// TIA Portal V16 export
// export: Created 2022-09-01T14:29:20.4817445Z, ExportSetting WithDefaults, DisplayName Totally Integrated Automation Portal, DisplayVersion V16, DisplayName TIA Portal Version Control Interface, DisplayVersion V16, DisplayName TIA Portal Openness, DisplayVersion V16, DisplayName STEP 7 Professional, DisplayVersion V16, DisplayName STEP 7 Safety, DisplayVersion V16, DisplayName WinCC Advanced, DisplayVersion V16
FUNCTION "Saídas" : Void   // FC2, LAD
{ S7_Optimized_Access := 'TRUE' }
VERSION : 0.1
// stored: AutoNumber true, IsIECCheckEnabled false, SetENOAutomatically false, UDAEnableTagReadback false
   VAR_TEMP   // added for the SCL form of the ladder/FBD networks
      _w1 : Bool;
   END_VAR
BEGIN

REGION Network 1: bomba de alimentação ao processo BS001A
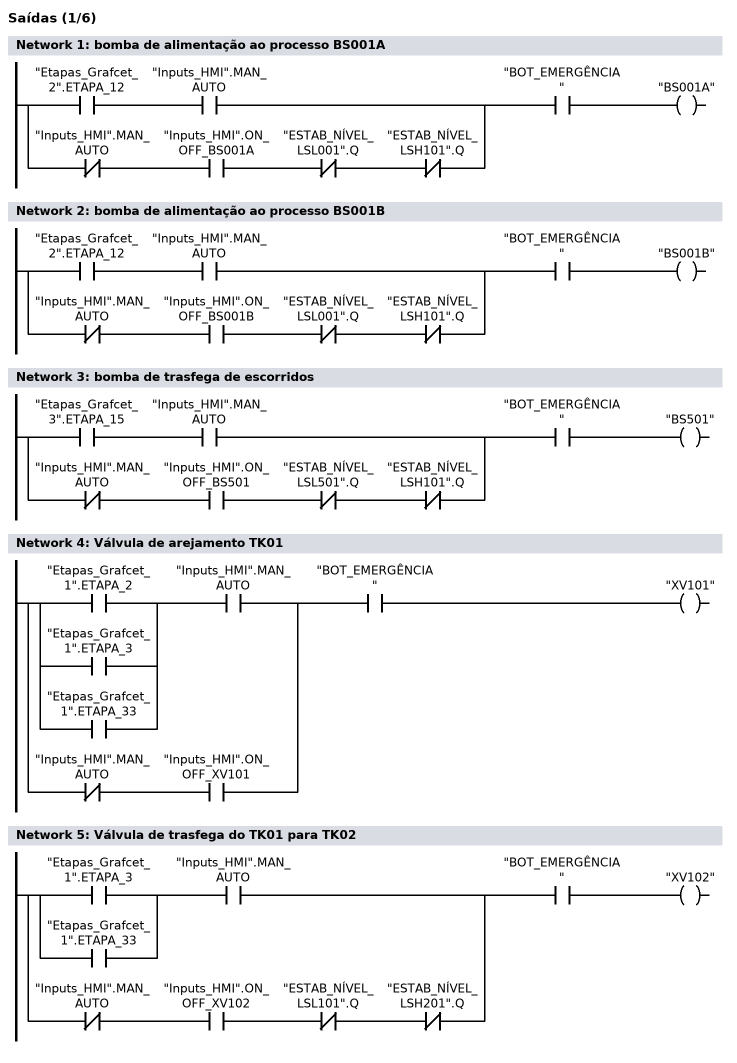
   RUNG wire#powerrail
      Contact( "Etapas_Grafcet_2".ETAPA_12 )
      Contact( "Inputs_HMI".MAN_AUTO )
      wire#w1
      Contact( "BOT_EMERGÊNCIA" )
      Coil( "BS001A" )
   END_RUNG
   RUNG wire#powerrail
      I_Contact( "Inputs_HMI".MAN_AUTO )
      Contact( "Inputs_HMI".ON_OFF_BS001A )
      I_Contact( "ESTAB_NÍVEL_LSL001".Q )
      I_Contact( "ESTAB_NÍVEL_LSH101".Q )
   END_RUNG wire#w1
   // the same network as SCL:
   "BS001A" := (("Etapas_Grafcet_2".ETAPA_12 AND "Inputs_HMI".MAN_AUTO) OR (NOT "Inputs_HMI".MAN_AUTO AND "Inputs_HMI".ON_OFF_BS001A AND NOT "ESTAB_NÍVEL_LSL001".Q AND NOT "ESTAB_NÍVEL_LSH101".Q)) AND "BOT_EMERGÊNCIA";
END_REGION

REGION Network 2: bomba de alimentação ao processo BS001B
   RUNG wire#powerrail
      Contact( "Etapas_Grafcet_2".ETAPA_12 )
      Contact( "Inputs_HMI".MAN_AUTO )
      wire#w1
      Contact( "BOT_EMERGÊNCIA" )
      Coil( "BS001B" )
   END_RUNG
   RUNG wire#powerrail
      I_Contact( "Inputs_HMI".MAN_AUTO )
      Contact( "Inputs_HMI".ON_OFF_BS001B )
      I_Contact( "ESTAB_NÍVEL_LSL001".Q )
      I_Contact( "ESTAB_NÍVEL_LSH101".Q )
   END_RUNG wire#w1
   // the same network as SCL:
   "BS001B" := (("Etapas_Grafcet_2".ETAPA_12 AND "Inputs_HMI".MAN_AUTO) OR (NOT "Inputs_HMI".MAN_AUTO AND "Inputs_HMI".ON_OFF_BS001B AND NOT "ESTAB_NÍVEL_LSL001".Q AND NOT "ESTAB_NÍVEL_LSH101".Q)) AND "BOT_EMERGÊNCIA";
END_REGION

REGION Network 3: bomba de trasfega de escorridos
   RUNG wire#powerrail
      Contact( "Etapas_Grafcet_3".ETAPA_15 )
      Contact( "Inputs_HMI".MAN_AUTO )
      wire#w1
      Contact( "BOT_EMERGÊNCIA" )
      Coil( "BS501" )
   END_RUNG
   RUNG wire#powerrail
      I_Contact( "Inputs_HMI".MAN_AUTO )
      Contact( "Inputs_HMI".ON_OFF_BS501 )
      I_Contact( "ESTAB_NÍVEL_LSL501".Q )
      I_Contact( "ESTAB_NÍVEL_LSH101".Q )
   END_RUNG wire#w1
   // the same network as SCL:
   "BS501" := (("Etapas_Grafcet_3".ETAPA_15 AND "Inputs_HMI".MAN_AUTO) OR (NOT "Inputs_HMI".MAN_AUTO AND "Inputs_HMI".ON_OFF_BS501 AND NOT "ESTAB_NÍVEL_LSL501".Q AND NOT "ESTAB_NÍVEL_LSH101".Q)) AND "BOT_EMERGÊNCIA";
END_REGION

REGION Network 4: Válvula de arejamento TK01
   RUNG wire#powerrail
      Contact( "Etapas_Grafcet_1".ETAPA_2 )
      wire#w1
      Contact( "Inputs_HMI".MAN_AUTO )
      wire#w2
      Contact( "BOT_EMERGÊNCIA" )
      Coil( "XV101" )
   END_RUNG
   RUNG wire#powerrail
      Contact( "Etapas_Grafcet_1".ETAPA_3 )
   END_RUNG wire#w1
   RUNG wire#powerrail
      Contact( "Etapas_Grafcet_1".ETAPA_33 )
   END_RUNG wire#w1
   RUNG wire#powerrail
      I_Contact( "Inputs_HMI".MAN_AUTO )
      Contact( "Inputs_HMI".ON_OFF_XV101 )
   END_RUNG wire#w2
   // the same network as SCL:
   "XV101" := ((("Etapas_Grafcet_1".ETAPA_2 OR "Etapas_Grafcet_1".ETAPA_3 OR "Etapas_Grafcet_1".ETAPA_33) AND "Inputs_HMI".MAN_AUTO) OR (NOT "Inputs_HMI".MAN_AUTO AND "Inputs_HMI".ON_OFF_XV101)) AND "BOT_EMERGÊNCIA";
END_REGION

REGION Network 5: Válvula de trasfega do TK01 para TK02
   RUNG wire#powerrail
      Contact( "Etapas_Grafcet_1".ETAPA_3 )
      wire#w1
      Contact( "Inputs_HMI".MAN_AUTO )
      wire#w2
      Contact( "BOT_EMERGÊNCIA" )
      Coil( "XV102" )
   END_RUNG
   RUNG wire#powerrail
      Contact( "Etapas_Grafcet_1".ETAPA_33 )
   END_RUNG wire#w1
   RUNG wire#powerrail
      I_Contact( "Inputs_HMI".MAN_AUTO )
      Contact( "Inputs_HMI".ON_OFF_XV102 )
      I_Contact( "ESTAB_NÍVEL_LSL101".Q )
      I_Contact( "ESTAB_NÍVEL_LSH201".Q )
   END_RUNG wire#w2
   // the same network as SCL:
   "XV102" := ((("Etapas_Grafcet_1".ETAPA_3 OR "Etapas_Grafcet_1".ETAPA_33) AND "Inputs_HMI".MAN_AUTO) OR (NOT "Inputs_HMI".MAN_AUTO AND "Inputs_HMI".ON_OFF_XV102 AND NOT "ESTAB_NÍVEL_LSL101".Q AND NOT "ESTAB_NÍVEL_LSH201".Q)) AND "BOT_EMERGÊNCIA";
END_REGION

REGION Network 6: Agitador MX201
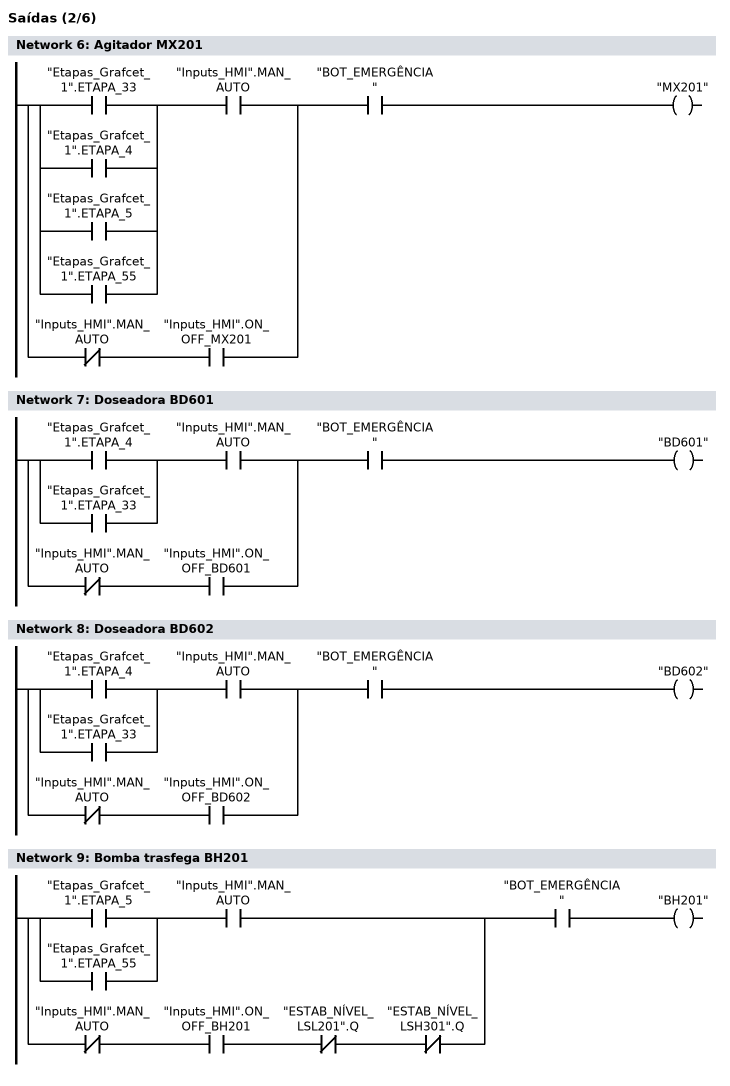
   RUNG wire#powerrail
      Contact( "Etapas_Grafcet_1".ETAPA_33 )
      wire#w1
      Contact( "Inputs_HMI".MAN_AUTO )
      wire#w2
      Contact( "BOT_EMERGÊNCIA" )
      Coil( "MX201" )
   END_RUNG
   RUNG wire#powerrail
      Contact( "Etapas_Grafcet_1".ETAPA_4 )
   END_RUNG wire#w1
   RUNG wire#powerrail
      Contact( "Etapas_Grafcet_1".ETAPA_5 )
   END_RUNG wire#w1
   RUNG wire#powerrail
      Contact( "Etapas_Grafcet_1".ETAPA_55 )
   END_RUNG wire#w1
   RUNG wire#powerrail
      I_Contact( "Inputs_HMI".MAN_AUTO )
      Contact( "Inputs_HMI".ON_OFF_MX201 )
   END_RUNG wire#w2
   // the same network as SCL:
   "MX201" := ((("Etapas_Grafcet_1".ETAPA_33 OR "Etapas_Grafcet_1".ETAPA_4 OR "Etapas_Grafcet_1".ETAPA_5 OR "Etapas_Grafcet_1".ETAPA_55) AND "Inputs_HMI".MAN_AUTO) OR (NOT "Inputs_HMI".MAN_AUTO AND "Inputs_HMI".ON_OFF_MX201)) AND "BOT_EMERGÊNCIA";
END_REGION

REGION Network 7: Doseadora BD601
   RUNG wire#powerrail
      Contact( "Etapas_Grafcet_1".ETAPA_4 )
      wire#w1
      Contact( "Inputs_HMI".MAN_AUTO )
      wire#w2
      Contact( "BOT_EMERGÊNCIA" )
      Coil( "BD601" )
   END_RUNG
   RUNG wire#powerrail
      Contact( "Etapas_Grafcet_1".ETAPA_33 )
   END_RUNG wire#w1
   RUNG wire#powerrail
      I_Contact( "Inputs_HMI".MAN_AUTO )
      Contact( "Inputs_HMI".ON_OFF_BD601 )
   END_RUNG wire#w2
   // the same network as SCL:
   "BD601" := ((("Etapas_Grafcet_1".ETAPA_4 OR "Etapas_Grafcet_1".ETAPA_33) AND "Inputs_HMI".MAN_AUTO) OR (NOT "Inputs_HMI".MAN_AUTO AND "Inputs_HMI".ON_OFF_BD601)) AND "BOT_EMERGÊNCIA";
END_REGION

REGION Network 8: Doseadora BD602
   RUNG wire#powerrail
      Contact( "Etapas_Grafcet_1".ETAPA_4 )
      wire#w1
      Contact( "Inputs_HMI".MAN_AUTO )
      wire#w2
      Contact( "BOT_EMERGÊNCIA" )
      Coil( "BD602" )
   END_RUNG
   RUNG wire#powerrail
      Contact( "Etapas_Grafcet_1".ETAPA_33 )
   END_RUNG wire#w1
   RUNG wire#powerrail
      I_Contact( "Inputs_HMI".MAN_AUTO )
      Contact( "Inputs_HMI".ON_OFF_BD602 )
   END_RUNG wire#w2
   // the same network as SCL:
   "BD602" := ((("Etapas_Grafcet_1".ETAPA_4 OR "Etapas_Grafcet_1".ETAPA_33) AND "Inputs_HMI".MAN_AUTO) OR (NOT "Inputs_HMI".MAN_AUTO AND "Inputs_HMI".ON_OFF_BD602)) AND "BOT_EMERGÊNCIA";
END_REGION

REGION Network 9: Bomba trasfega BH201
   RUNG wire#powerrail
      Contact( "Etapas_Grafcet_1".ETAPA_5 )
      wire#w1
      Contact( "Inputs_HMI".MAN_AUTO )
      wire#w2
      Contact( "BOT_EMERGÊNCIA" )
      Coil( "BH201" )
   END_RUNG
   RUNG wire#powerrail
      Contact( "Etapas_Grafcet_1".ETAPA_55 )
   END_RUNG wire#w1
   RUNG wire#powerrail
      I_Contact( "Inputs_HMI".MAN_AUTO )
      Contact( "Inputs_HMI".ON_OFF_BH201 )
      I_Contact( "ESTAB_NÍVEL_LSL201".Q )
      I_Contact( "ESTAB_NÍVEL_LSH301".Q )
   END_RUNG wire#w2
   // the same network as SCL:
   "BH201" := ((("Etapas_Grafcet_1".ETAPA_5 OR "Etapas_Grafcet_1".ETAPA_55) AND "Inputs_HMI".MAN_AUTO) OR (NOT "Inputs_HMI".MAN_AUTO AND "Inputs_HMI".ON_OFF_BH201 AND NOT "ESTAB_NÍVEL_LSL201".Q AND NOT "ESTAB_NÍVEL_LSH301".Q)) AND "BOT_EMERGÊNCIA";
END_REGION

REGION Network 10: Agitador MX301
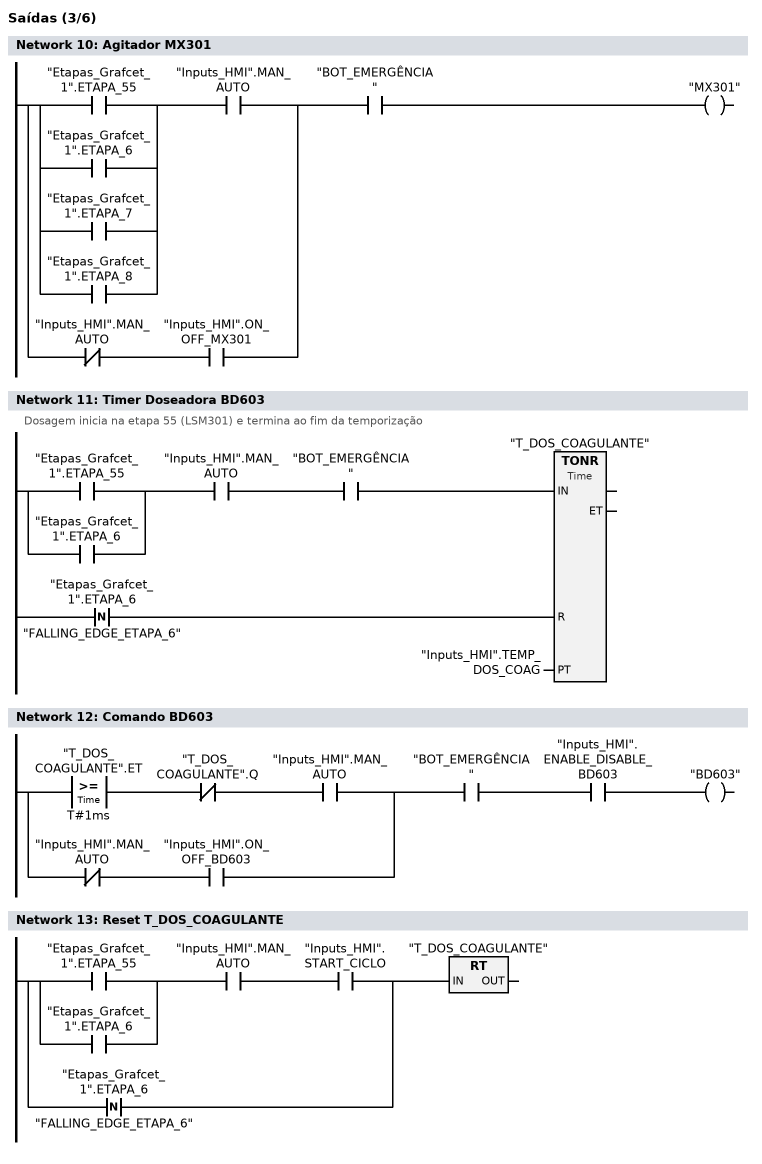
   RUNG wire#powerrail
      Contact( "Etapas_Grafcet_1".ETAPA_55 )
      wire#w1
      Contact( "Inputs_HMI".MAN_AUTO )
      wire#w2
      Contact( "BOT_EMERGÊNCIA" )
      Coil( "MX301" )
   END_RUNG
   RUNG wire#powerrail
      Contact( "Etapas_Grafcet_1".ETAPA_6 )
   END_RUNG wire#w1
   RUNG wire#powerrail
      Contact( "Etapas_Grafcet_1".ETAPA_7 )
   END_RUNG wire#w1
   RUNG wire#powerrail
      Contact( "Etapas_Grafcet_1".ETAPA_8 )
   END_RUNG wire#w1
   RUNG wire#powerrail
      I_Contact( "Inputs_HMI".MAN_AUTO )
      Contact( "Inputs_HMI".ON_OFF_MX301 )
   END_RUNG wire#w2
   // the same network as SCL:
   "MX301" := ((("Etapas_Grafcet_1".ETAPA_55 OR "Etapas_Grafcet_1".ETAPA_6 OR "Etapas_Grafcet_1".ETAPA_7 OR "Etapas_Grafcet_1".ETAPA_8) AND "Inputs_HMI".MAN_AUTO) OR (NOT "Inputs_HMI".MAN_AUTO AND "Inputs_HMI".ON_OFF_MX301)) AND "BOT_EMERGÊNCIA";
END_REGION

REGION Network 11: Timer Doseadora BD603
   // Dosagem inicia na etapa 55 (LSM301) e termina ao fim da temporização
   RUNG wire#powerrail
      Contact( "Etapas_Grafcet_1".ETAPA_55 )
      wire#w1
      Contact( "Inputs_HMI".MAN_AUTO )
      Contact( "BOT_EMERGÊNCIA" )
      { S7_Templates := "time_type := Time" } "T_DOS_COAGULANTE".TONR(r := wire#w2, pt := "Inputs_HMI".TEMP_DOS_COAG, et =>)
   END_RUNG
   RUNG wire#powerrail
      Contact( "Etapas_Grafcet_1".ETAPA_6 )
   END_RUNG wire#w1
   RUNG wire#powerrail
      N_Contact(operand := "Etapas_Grafcet_1".ETAPA_6, bit := "FALLING_EDGE_ETAPA_6")
   END_RUNG wire#w2
   // the same network as SCL:
   #_w1 := NOT "Etapas_Grafcet_1".ETAPA_6 AND "FALLING_EDGE_ETAPA_6";   // falling edge of "Etapas_Grafcet_1".ETAPA_6
   "FALLING_EDGE_ETAPA_6" := "Etapas_Grafcet_1".ETAPA_6;
   "T_DOS_COAGULANTE".TONR(IN := ("Etapas_Grafcet_1".ETAPA_55 OR "Etapas_Grafcet_1".ETAPA_6) AND "Inputs_HMI".MAN_AUTO AND "BOT_EMERGÊNCIA",
                           R := #_w1,
                           PT := "Inputs_HMI".TEMP_DOS_COAG);
END_REGION

REGION Network 12: Comando BD603
   RUNG wire#powerrail
      { S7_Templates := "SrcType := Time" } GE_Contact(in1 := "T_DOS_COAGULANTE".ET, in2 := T#1ms)
      I_Contact( "T_DOS_COAGULANTE".Q )
      Contact( "Inputs_HMI".MAN_AUTO )
      wire#w1
      Contact( "BOT_EMERGÊNCIA" )
      Contact( "Inputs_HMI".ENABLE_DISABLE_BD603 )
      Coil( "BD603" )
   END_RUNG
   RUNG wire#powerrail
      I_Contact( "Inputs_HMI".MAN_AUTO )
      Contact( "Inputs_HMI".ON_OFF_BD603 )
   END_RUNG wire#w1
   // the same network as SCL:
   "BD603" := ((("T_DOS_COAGULANTE".ET >= T#1ms) AND NOT "T_DOS_COAGULANTE".Q AND "Inputs_HMI".MAN_AUTO) OR (NOT "Inputs_HMI".MAN_AUTO AND "Inputs_HMI".ON_OFF_BD603)) AND "BOT_EMERGÊNCIA" AND "Inputs_HMI".ENABLE_DISABLE_BD603;
END_REGION

REGION Network 13: Reset T_DOS_COAGULANTE
   RUNG wire#powerrail
      Contact( "Etapas_Grafcet_1".ETAPA_55 )
      wire#w1
      Contact( "Inputs_HMI".MAN_AUTO )
      Contact( "Inputs_HMI".START_CICLO )
      wire#w2
      RT_Coil( "T_DOS_COAGULANTE" )
   END_RUNG
   RUNG wire#powerrail
      Contact( "Etapas_Grafcet_1".ETAPA_6 )
   END_RUNG wire#w1
   RUNG wire#powerrail
      N_Contact(operand := "Etapas_Grafcet_1".ETAPA_6, bit := "FALLING_EDGE_ETAPA_6")
   END_RUNG wire#w2
   // the same network as SCL:
   #_w1 := NOT "Etapas_Grafcet_1".ETAPA_6 AND "FALLING_EDGE_ETAPA_6";   // falling edge of "Etapas_Grafcet_1".ETAPA_6
   "FALLING_EDGE_ETAPA_6" := "Etapas_Grafcet_1".ETAPA_6;
   IF (("Etapas_Grafcet_1".ETAPA_55 OR "Etapas_Grafcet_1".ETAPA_6) AND "Inputs_HMI".MAN_AUTO AND "Inputs_HMI".START_CICLO) OR #_w1 THEN
       RESET_TIMER("T_DOS_COAGULANTE");
   END_IF;
END_REGION

REGION Network 14: Doseadora BD604
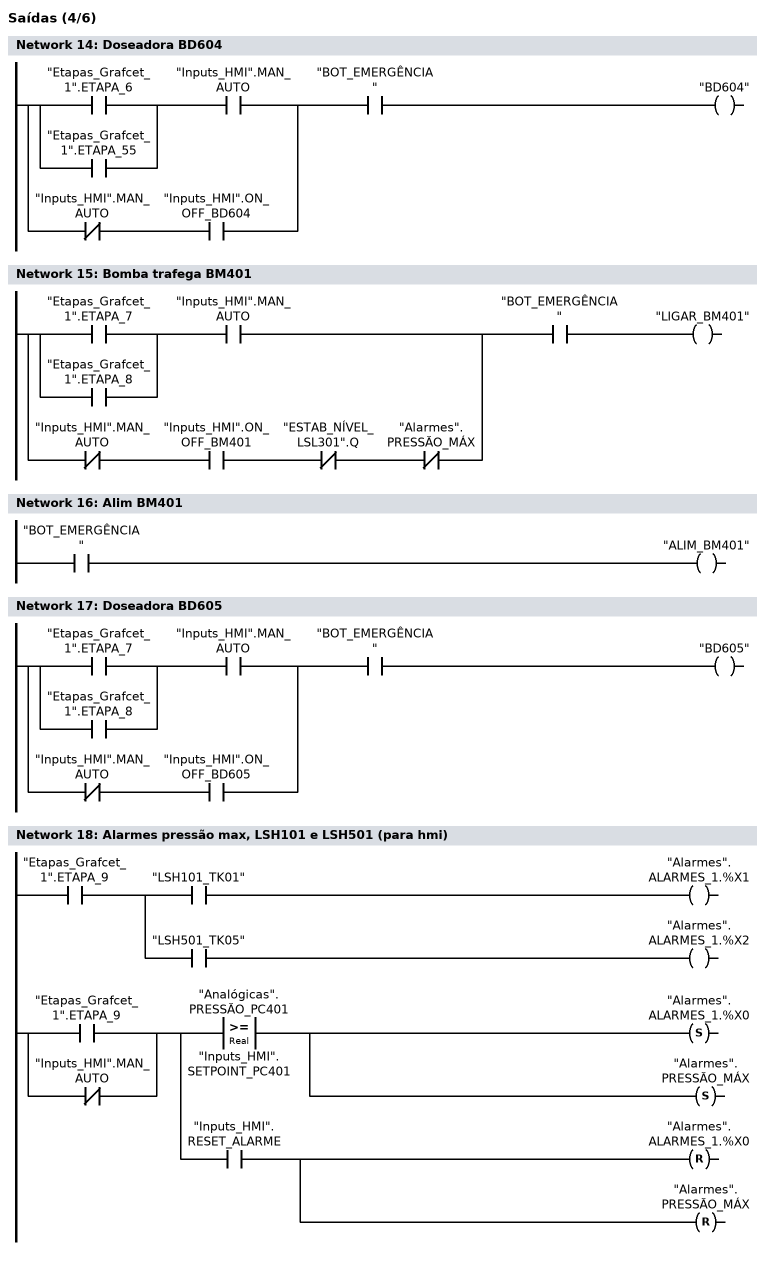
   RUNG wire#powerrail
      Contact( "Etapas_Grafcet_1".ETAPA_6 )
      wire#w1
      Contact( "Inputs_HMI".MAN_AUTO )
      wire#w2
      Contact( "BOT_EMERGÊNCIA" )
      Coil( "BD604" )
   END_RUNG
   RUNG wire#powerrail
      Contact( "Etapas_Grafcet_1".ETAPA_55 )
   END_RUNG wire#w1
   RUNG wire#powerrail
      I_Contact( "Inputs_HMI".MAN_AUTO )
      Contact( "Inputs_HMI".ON_OFF_BD604 )
   END_RUNG wire#w2
   // the same network as SCL:
   "BD604" := ((("Etapas_Grafcet_1".ETAPA_6 OR "Etapas_Grafcet_1".ETAPA_55) AND "Inputs_HMI".MAN_AUTO) OR (NOT "Inputs_HMI".MAN_AUTO AND "Inputs_HMI".ON_OFF_BD604)) AND "BOT_EMERGÊNCIA";
END_REGION

REGION Network 15: Bomba trafega BM401
   RUNG wire#powerrail
      Contact( "Etapas_Grafcet_1".ETAPA_7 )
      wire#w1
      Contact( "Inputs_HMI".MAN_AUTO )
      wire#w2
      Contact( "BOT_EMERGÊNCIA" )
      Coil( "LIGAR_BM401" )
   END_RUNG
   RUNG wire#powerrail
      Contact( "Etapas_Grafcet_1".ETAPA_8 )
   END_RUNG wire#w1
   RUNG wire#powerrail
      I_Contact( "Inputs_HMI".MAN_AUTO )
      Contact( "Inputs_HMI".ON_OFF_BM401 )
      I_Contact( "ESTAB_NÍVEL_LSL301".Q )
      I_Contact( "Alarmes".PRESSÃO_MÁX )
   END_RUNG wire#w2
   // the same network as SCL:
   "LIGAR_BM401" := ((("Etapas_Grafcet_1".ETAPA_7 OR "Etapas_Grafcet_1".ETAPA_8) AND "Inputs_HMI".MAN_AUTO) OR (NOT "Inputs_HMI".MAN_AUTO AND "Inputs_HMI".ON_OFF_BM401 AND NOT "ESTAB_NÍVEL_LSL301".Q AND NOT "Alarmes".PRESSÃO_MÁX)) AND "BOT_EMERGÊNCIA";
END_REGION

REGION Network 16: Alim BM401
   RUNG wire#powerrail
      Contact( "BOT_EMERGÊNCIA" )
      Coil( "ALIM_BM401" )
   END_RUNG
   // the same network as SCL:
   "ALIM_BM401" := "BOT_EMERGÊNCIA";
END_REGION

REGION Network 17: Doseadora BD605
   RUNG wire#powerrail
      Contact( "Etapas_Grafcet_1".ETAPA_7 )
      wire#w1
      Contact( "Inputs_HMI".MAN_AUTO )
      wire#w2
      Contact( "BOT_EMERGÊNCIA" )
      Coil( "BD605" )
   END_RUNG
   RUNG wire#powerrail
      Contact( "Etapas_Grafcet_1".ETAPA_8 )
   END_RUNG wire#w1
   RUNG wire#powerrail
      I_Contact( "Inputs_HMI".MAN_AUTO )
      Contact( "Inputs_HMI".ON_OFF_BD605 )
   END_RUNG wire#w2
   // the same network as SCL:
   "BD605" := ((("Etapas_Grafcet_1".ETAPA_7 OR "Etapas_Grafcet_1".ETAPA_8) AND "Inputs_HMI".MAN_AUTO) OR (NOT "Inputs_HMI".MAN_AUTO AND "Inputs_HMI".ON_OFF_BD605)) AND "BOT_EMERGÊNCIA";
END_REGION

REGION Network 18: Alarmes pressão max, LSH101 e LSH501 (para hmi)
   RUNG wire#powerrail
      Contact( "Etapas_Grafcet_1".ETAPA_9 )
      wire#w1
      Contact( "LSH101_TK01" )
      Coil( "Alarmes".ALARMES_1.%X1 )
   END_RUNG
   RUNG wire#w1
      Contact( "LSH501_TK05" )
      Coil( "Alarmes".ALARMES_1.%X2 )
   END_RUNG
   RUNG wire#powerrail
      Contact( "Etapas_Grafcet_1".ETAPA_9 )
      wire#w2
      { S7_Templates := "SrcType := Real" } GE_Contact(in1 := "Analógicas".PRESSÃO_PC401, in2 := "Inputs_HMI".SETPOINT_PC401)
      wire#w3
      S_Coil( "Alarmes".ALARMES_1.%X0 )
   END_RUNG
   RUNG wire#powerrail
      I_Contact( "Inputs_HMI".MAN_AUTO )
   END_RUNG wire#w2
   RUNG wire#w3
      S_Coil( "Alarmes".PRESSÃO_MÁX )
   END_RUNG
   RUNG wire#w2
      Contact( "Inputs_HMI".RESET_ALARME )
      wire#w4
      R_Coil( "Alarmes".ALARMES_1.%X0 )
   END_RUNG
   RUNG wire#w4
      R_Coil( "Alarmes".PRESSÃO_MÁX )
   END_RUNG
   // the same network as SCL:
   "Alarmes".ALARMES_1.%X1 := "Etapas_Grafcet_1".ETAPA_9 AND "LSH101_TK01";
   "Alarmes".ALARMES_1.%X2 := "Etapas_Grafcet_1".ETAPA_9 AND "LSH501_TK05";
   #_w1 := "Etapas_Grafcet_1".ETAPA_9 OR NOT "Inputs_HMI".MAN_AUTO;
   IF #_w1 AND ("Analógicas".PRESSÃO_PC401 >= "Inputs_HMI".SETPOINT_PC401) THEN
       "Alarmes".ALARMES_1.%X0 := TRUE;
       "Alarmes".PRESSÃO_MÁX := TRUE;
   END_IF;
   IF #_w1 AND "Inputs_HMI".RESET_ALARME THEN
       "Alarmes".ALARMES_1.%X0 := FALSE;
       "Alarmes".PRESSÃO_MÁX := FALSE;
   END_IF;
END_REGION

REGION Network 19: Alarme (luminoso)
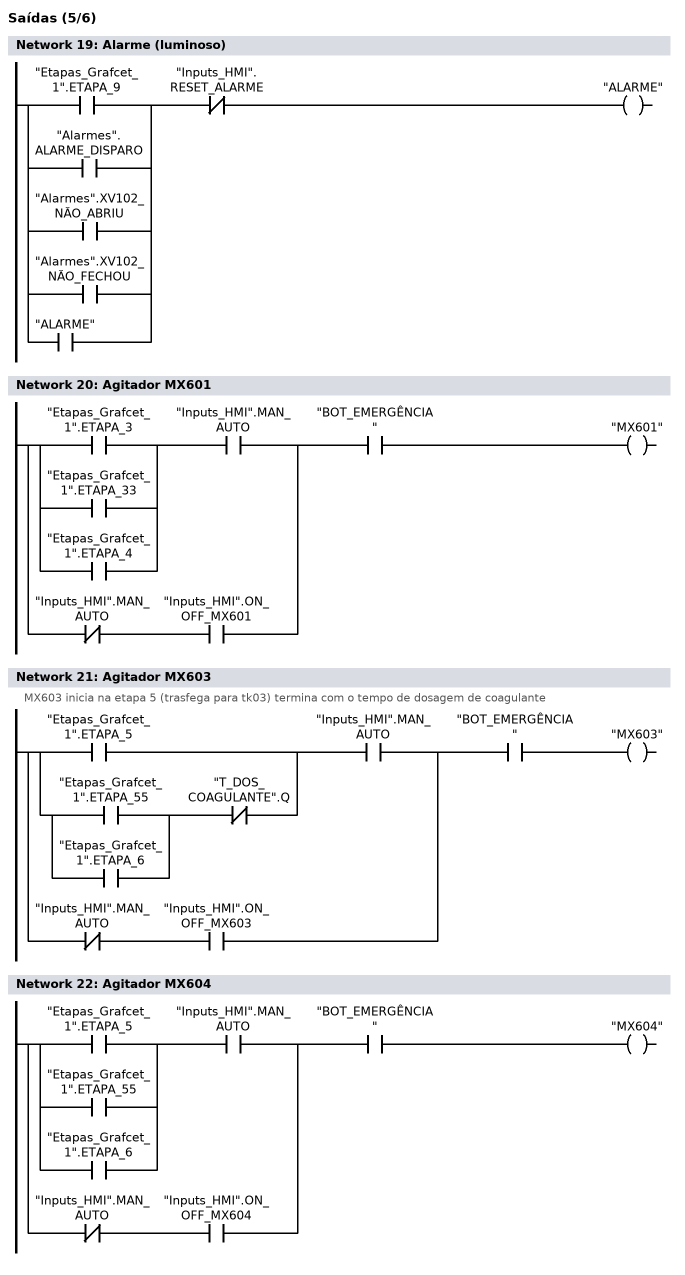
   RUNG wire#powerrail
      Contact( "Etapas_Grafcet_1".ETAPA_9 )
      wire#w1
      I_Contact( "Inputs_HMI".RESET_ALARME )
      Coil( "ALARME" )
   END_RUNG
   RUNG wire#powerrail
      Contact( "Alarmes".ALARME_DISPARO )
   END_RUNG wire#w1
   RUNG wire#powerrail
      Contact( "Alarmes".XV102_NÃO_ABRIU )
   END_RUNG wire#w1
   RUNG wire#powerrail
      Contact( "Alarmes".XV102_NÃO_FECHOU )
   END_RUNG wire#w1
   RUNG wire#powerrail
      Contact( "ALARME" )
   END_RUNG wire#w1
   // the same network as SCL:
   "ALARME" := ("Etapas_Grafcet_1".ETAPA_9 OR "Alarmes".ALARME_DISPARO OR "Alarmes".XV102_NÃO_ABRIU OR "Alarmes".XV102_NÃO_FECHOU OR "ALARME") AND NOT "Inputs_HMI".RESET_ALARME;
END_REGION

REGION Network 20: Agitador MX601
   RUNG wire#powerrail
      Contact( "Etapas_Grafcet_1".ETAPA_3 )
      wire#w1
      Contact( "Inputs_HMI".MAN_AUTO )
      wire#w2
      Contact( "BOT_EMERGÊNCIA" )
      Coil( "MX601" )
   END_RUNG
   RUNG wire#powerrail
      Contact( "Etapas_Grafcet_1".ETAPA_33 )
   END_RUNG wire#w1
   RUNG wire#powerrail
      Contact( "Etapas_Grafcet_1".ETAPA_4 )
   END_RUNG wire#w1
   RUNG wire#powerrail
      I_Contact( "Inputs_HMI".MAN_AUTO )
      Contact( "Inputs_HMI".ON_OFF_MX601 )
   END_RUNG wire#w2
   // the same network as SCL:
   "MX601" := ((("Etapas_Grafcet_1".ETAPA_3 OR "Etapas_Grafcet_1".ETAPA_33 OR "Etapas_Grafcet_1".ETAPA_4) AND "Inputs_HMI".MAN_AUTO) OR (NOT "Inputs_HMI".MAN_AUTO AND "Inputs_HMI".ON_OFF_MX601)) AND "BOT_EMERGÊNCIA";
END_REGION

REGION Network 21: Agitador MX603
   // MX603 inicia na etapa 5 (trasfega para tk03) termina com o tempo de dosagem de coagulante
   RUNG wire#powerrail
      Contact( "Etapas_Grafcet_1".ETAPA_5 )
      wire#w1
      Contact( "Inputs_HMI".MAN_AUTO )
      wire#w3
      Contact( "BOT_EMERGÊNCIA" )
      Coil( "MX603" )
   END_RUNG
   RUNG wire#powerrail
      Contact( "Etapas_Grafcet_1".ETAPA_55 )
      wire#w2
      I_Contact( "T_DOS_COAGULANTE".Q )
   END_RUNG wire#w1
   RUNG wire#powerrail
      Contact( "Etapas_Grafcet_1".ETAPA_6 )
   END_RUNG wire#w2
   RUNG wire#powerrail
      I_Contact( "Inputs_HMI".MAN_AUTO )
      Contact( "Inputs_HMI".ON_OFF_MX603 )
   END_RUNG wire#w3
   // the same network as SCL:
   "MX603" := ((("Etapas_Grafcet_1".ETAPA_5 OR (("Etapas_Grafcet_1".ETAPA_55 OR "Etapas_Grafcet_1".ETAPA_6) AND NOT "T_DOS_COAGULANTE".Q)) AND "Inputs_HMI".MAN_AUTO) OR (NOT "Inputs_HMI".MAN_AUTO AND "Inputs_HMI".ON_OFF_MX603)) AND "BOT_EMERGÊNCIA";
END_REGION

REGION Network 22: Agitador MX604
   RUNG wire#powerrail
      Contact( "Etapas_Grafcet_1".ETAPA_5 )
      wire#w1
      Contact( "Inputs_HMI".MAN_AUTO )
      wire#w2
      Contact( "BOT_EMERGÊNCIA" )
      Coil( "MX604" )
   END_RUNG
   RUNG wire#powerrail
      Contact( "Etapas_Grafcet_1".ETAPA_55 )
   END_RUNG wire#w1
   RUNG wire#powerrail
      Contact( "Etapas_Grafcet_1".ETAPA_6 )
   END_RUNG wire#w1
   RUNG wire#powerrail
      I_Contact( "Inputs_HMI".MAN_AUTO )
      Contact( "Inputs_HMI".ON_OFF_MX604 )
   END_RUNG wire#w2
   // the same network as SCL:
   "MX604" := ((("Etapas_Grafcet_1".ETAPA_5 OR "Etapas_Grafcet_1".ETAPA_55 OR "Etapas_Grafcet_1".ETAPA_6) AND "Inputs_HMI".MAN_AUTO) OR (NOT "Inputs_HMI".MAN_AUTO AND "Inputs_HMI".ON_OFF_MX604)) AND "BOT_EMERGÊNCIA";
END_REGION

REGION Network 23: Agitador MX605
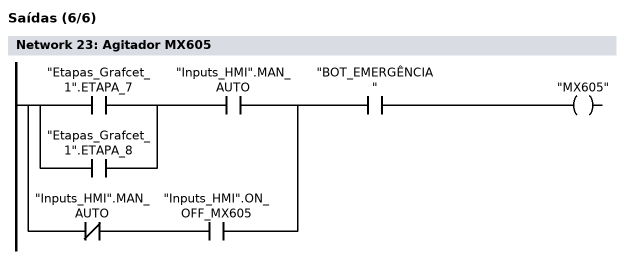
   RUNG wire#powerrail
      Contact( "Etapas_Grafcet_1".ETAPA_7 )
      wire#w1
      Contact( "Inputs_HMI".MAN_AUTO )
      wire#w2
      Contact( "BOT_EMERGÊNCIA" )
      Coil( "MX605" )
   END_RUNG
   RUNG wire#powerrail
      Contact( "Etapas_Grafcet_1".ETAPA_8 )
   END_RUNG wire#w1
   RUNG wire#powerrail
      I_Contact( "Inputs_HMI".MAN_AUTO )
      Contact( "Inputs_HMI".ON_OFF_MX605 )
   END_RUNG wire#w2
   // the same network as SCL:
   "MX605" := ((("Etapas_Grafcet_1".ETAPA_7 OR "Etapas_Grafcet_1".ETAPA_8) AND "Inputs_HMI".MAN_AUTO) OR (NOT "Inputs_HMI".MAN_AUTO AND "Inputs_HMI".ON_OFF_MX605)) AND "BOT_EMERGÊNCIA";
END_REGION
END_FUNCTION
